// TIA Portal project "Program_PLC" (V15.1)

(* hardware
DEVICE "S7-1200"  S7-1200 Station
   slot 0: "Rack_0"  S7-1200 Rack  Rack  V1.0
   slot 1: "PLC1"  CPU 1215C AC/DC/Rly  6ES7 215-1BG40-0XB0  V4.2
*)

// ===== PLC "PLC1"  CPU 1215C AC/DC/Rly =====

VAR_GLOBAL   // PLC tag table "Default tag table"
   "Clock_Byte" AT %MB0 : Byte;   // Clock_Byte
   "Clock_10Hz" AT %M0.0 : Bool;   // Clock_10Hz
   "Clock_5Hz" AT %M0.1 : Bool;   // Clock_5Hz
   "Clock_2.5Hz" AT %M0.2 : Bool;   // Clock_2.5Hz
   "Clock_2Hz" AT %M0.3 : Bool;   // Clock_2Hz
   "Clock_1.25Hz" AT %M0.4 : Bool;   // Clock_1.25Hz
   "Clock_1Hz" AT %M0.5 : Bool;   // Clock_1Hz
   "Clock_0.625Hz" AT %M0.6 : Bool;   // Clock_0.625Hz
   "Clock_0.5Hz" AT %M0.7 : Bool;   // Clock_0.5Hz
   "System_Byte" AT %MB1 : Byte;   // System_Byte
   "FirstScan" AT %M1.0 : Bool;   // FirstScan
   "DiagStatusUpdate" AT %M1.1 : Bool;   // DiagStatusUpdate
   "AlwaysTRUE" AT %M1.2 : Bool;   // Sempre Um
   "AlwaysFALSE" AT %M1.3 : Bool;   // Sempre Zero
END_VAR

// folder: DB

DATA_BLOCK "Dados_Snap7"   // DB3
{ S7_Optimized_Access := 'FALSE' }
VERSION : 0.1
   VAR
      Dados1 : Word;
      Dados2 : Word;
      Dados3 : Word;
      Dados4 : Word;
      Dados5 : Word;
      Dados6 : Word;
      Dados7 : Word;
      Dados8 : Word;
      Dados9 : Word;
      Dados10 : Word;
      Dados11 : Word;
      Dados12 : Word;
      Dados13 : Word;
      Dados14 : Word;
      Dados15 : Word;
      Dados16 : Word;
      Dados17 : Word;
      Dados18 : Word;
      Dados19 : Word;
      Dados20 : Word;
   END_VAR
BEGIN
END_DATA_BLOCK

// folder: System blocks/Program resources

DATA_BLOCK "Timer_fachar_portao"   // DB1
{ S7_Optimized_Access := 'TRUE' }
AUTHOR : Simatic
FAMILY : IEC
NAME : IEC_TMR
VERSION : 1.0
// stored: InstanceOfName IEC_TIMER
"IEC_TIMER"
BEGIN
END_DATA_BLOCK

DATA_BLOCK "IEC_Timer_0_DB"   // DB2
{ S7_Optimized_Access := 'TRUE' }
AUTHOR : Simatic
FAMILY : IEC
NAME : IEC_TMR
VERSION : 1.0
// stored: InstanceOfName IEC_TIMER
"IEC_TIMER"
BEGIN
END_DATA_BLOCK

// folder: (top level)

ORGANIZATION_BLOCK "Main"   // OB1, LAD, ProgramCycle
TITLE = "Main Program Sweep (Cycle)"
{ S7_Optimized_Access := 'TRUE' }
VERSION : 0.1
   VAR_INPUT
      Initial_Call : Bool;   // Initial call of this OB
      Remanence : Bool;   // =True, if remanent data are available
   END_VAR
BEGIN
END_ORGANIZATION_BLOCK